(* PLC project Cell Example , CTH FIX1 1.0, author CTH SS2 *)
(* stored: companyURL www.chalmers.se, creationDateTime 2008-03-19T20:31:26, version 1.0, modificationDateTime 2008-04-03T17:05:15, organization SS2, language en-US *)

FUNCTION_BLOCK RAC

(* LD diagram, written out as Structured Text *)
END_FUNCTION_BLOCK

CONFIGURATION ExampleCell
END_CONFIGURATION
